# EPICS autosave request: BPMApp/Db/BPMDsp_settings.req
$(P)$(R)PosKx-SP
$(P)$(R)PosKy-SP
$(P)$(R)PosKq-SP
$(P)$(R)PosKsum-SP
$(P)$(R)PosXOffset-SP
$(P)$(R)PosYOffset-SP
$(P)$(R)PosQOffset-SP
$(P)$(R)SwTagEn-Sel
$(P)$(R)SwDataMaskEn-Sel
$(P)$(R)SwDataMaskSamples-SP
$(P)$(R)TbtTagEn-Sel
$(P)$(R)TbtTagDly-Sel
$(P)$(R)TbtDataMaskEn-Sel
$(P)$(R)TbtDataMaskSamplesBeg-SP
$(P)$(R)TbtDataMaskSamplesEnd-SP
